(* CoDeSys 2.3 export: SELECTSCREENADDSTRUC.EXP *)

(* Data type in Other *)
TYPE SelectScreenAddStruc :
STRUCT
    strIn: STRING(5);    (*строка, дописываемая между ВЫХОД и ВХОД*)
END_STRUCT
END_TYPE
